TYPE EcCoeSdoRead_CMD_typ :
	STRUCT
		Enable	: BOOL ;
	END_STRUCT
END_TYPE

(* stored: Version 1.1.0.1, ProductVersion 3.1.4024.3
   DUT EcCoeSdoRead_CMD_typ: Id {a911d288-a02e-06c6-0f7b-61b7bc56a4f2} *)
